TYPE T_AVL_Map_Node : ST_AVL_MAP_NODE; END_TYPE

(* stored: Version 1.1.0.1
   DUT T_AVL_Map_Node: Id {074b8e2f-6a09-01a7-392c-4993822e0684} *)
